   // Fliegendes Referenzieren aktivieren erkennen
   IF #FlyRef AND NOT #sbRefTypEdge THEN
     #sbRefTyp := True;
   END_IF;
   // Fliegendes Referenzieren aktivieren Flanke merken
   #sbRefTypEdge := #FlyRef;

   // Fliegendes Referenzieren Flankenmerker wieder zurücksetzen
   IF NOT #FlyRef THEN
     #sbRefTyp := False;
     #siRefTypCyc := 0;
   END_IF;

   // Betriebsart aktivieren erkennen (RQ 3901129, RQ 4094299)
   IF #ExecuteMode AND NOT #sbExecuteEdge THEN
     #sbExecute := True;
     #siExecuteCyc := 0;
   ELSIF #ActMode <> #ModePos THEN
     #sbExecute := FALSE;
   ELSIF #siExecuteCyc > (2 * #siCycWait) THEN
     IF #ModePos <> 4 THEN
       #sbExecute := FALSE;
     ELSE
       IF #sxRecvBuf.ZSW1.%X11 OR NOT #ExecuteMode THEN
         #sbExecute := FALSE;
       END_IF;
     END_IF;
   ELSE
     ; // not used
   END_IF;

   IF #siExecuteCyc > 100 THEN
     #siExecuteCyc := 0;
   ELSE
     #siExecuteCyc := #siExecuteCyc + 1;
   END_IF;

   // Verfahrauftrag aktivieren Flanke merken
   #sbExecuteEdge := #ExecuteMode;

   // Betriebsart MDI / Sollwertdirektvorgabe Flanke merken
   (*IF #sxSendBuf.sxEPosSTW1.MdiStart AND NOT #sbMdiStartEdge THEN
             #sbMdiStart := True;
         END_IF;
         // Betriebsart MDI / Sollwertdirektvorgabe Flanke merken
         #sbMdiStartEdge := #sxSendBuf.sxEPosSTW1.MdiStart AND NOT #Busy;*)

   // Verfahrauftragflankenmerker wieder zurücksetzen
   (*IF NOT #sxSendBuf.sxEPosSTW1.MdiStart THEN
             #sbMdiStart := False;
             #siMdiStartCyc := 0;
         END_IF;*)

   IF #sxSendBuf.EPosSTW1.%X15 AND NOT #sbMdiStartEdge THEN
     #sbMdiStart := True;
   END_IF;
   // Betriebsart MDI / Sollwertdirektvorgabe Flanke merken
   #sbMdiStartEdge := #sxSendBuf.EPosSTW1.%X15 AND NOT #sbBusy;

   // Verfahrauftragflankenmerker wieder zurücksetzen
   IF NOT #sxSendBuf.EPosSTW1.%X15 THEN
     #sbMdiStart := False;
     #siMdiStartCyc := 0;
   END_IF;

   // Schreibdaten zusammenstellen
   // Steuerword STW1 für alle Betriebsart aufbereiten
   (*#sxSendBuf.sxSTW1.RejTrvTsk        := #RejTrvTsk;
         #sxSendBuf.sxSTW1.IntMStop         := #IntMStop;
         #sxSendBuf.sxSTW1.AckFault         := #AckFlt;*)

   #sxSendBuf.STW1.%X4 := #CancelTraversing;
   #sxSendBuf.STW1.%X5 := #IntermediateStop;
   #sxSendBuf.STW1.%X7 := #AckError;
   #sxSendBuf.STW1.%X1 := TRUE;
   #sxSendBuf.STW1.%X2 := TRUE;
   #sxSendBuf.STW1.%X3 := TRUE;
   #sxSendBuf.STW1.%X10 := TRUE;

   // Hauptbetriebsart "Positionieren / manueller Sollwertvorgabe (MDI)" 
   // Betriebsart "Positionieren Relativ positiv" oder "Positionieren Relativ negativ"
   IF (#siModePos = 1 AND #sbModePos) THEN

     // Antrieb einschalten
     //#sxSendBuf.sxSTW1.Off1 := #sbOff1;
     #sxSendBuf.STW1.%X0 := #sbOff1;

     // nicht verwendete Signale für den 1. Schritt und eventuell weitere Schritte
     (*#sxSendBuf.sxSTW1.Jog1          := False;
             #sxSendBuf.sxSTW1.Jog2          := False;
             #sxSendBuf.sxEPosSTW1.MdiTyp    := False;
             #sxSendBuf.sxEPosSTW1.MdiPos    := False;
             #sxSendBuf.sxEPosSTW1.MdiNeg    := False;
             #sxSendBuf.sxEPosSTW1.MdiSetup  := False;
             #sxSendBuf.sxEPosSTW2.SetRefPt  := False;
             #sxSendBuf.sxEPosSTW2.JogInc    := False;
             #sxSendBuf.sxEPosSTW2.RefStDi   := False;
             #sxSendBuf.sxSTW1.RefStart      := False;
             #sxSendBuf.sxEPosSTW2.RefTyp    := False;
             #sxSendBuf.sxEPosSTW1.MdiStart  := False;*)
     #sxSendBuf.STW1.%X8 := False;
     #sxSendBuf.STW1.%X9 := False;
     #sxSendBuf.EPosSTW1.%X8 := False;
     #sxSendBuf.EPosSTW1.%X9 := False;
     #sxSendBuf.EPosSTW1.%X10 := False;
     #sxSendBuf.EPosSTW1.%X14 := False;
     #sxSendBuf.EPosSTW2.%X1 := False;
     #sxSendBuf.EPosSTW2.%X5 := False;
     #sxSendBuf.EPosSTW2.%X9 := False;
     #sxSendBuf.STW1.%X11 := False;
     #sxSendBuf.EPosSTW2.%X8 := False;
     #sxSendBuf.EPosSTW1.%X15 := False;


     // Nach dem Einschalten des Antriebes, prüfen ob der Antrieb betriebsbereit, in Operation ohne Fehler und Warnung ist, 
     // dann die Betriebsart MDI / Sollwertvorgabe Start gesetzt werden
     IF #sbOff1 AND #sbReady AND #sbIOp AND NOT #sbFault THEN

       // Betriebsart MDI / Sollwertdirektvorgabe setzen
       //#sxSendBuf.sxEPosSTW1.MdiStart := True;
       #sxSendBuf.EPosSTW1.%X15 := True;

       // Positioniertyp auf relatives Positionieren stellen 
       //#sxSendBuf.sxEPosSTW1.MdiTyp := False;
       #sxSendBuf.EPosSTW1.%X8 := False;

       // die Richtungswahl für das Positionieren auf positive Richtung oder negative Richtung einstellen
       IF #Positive AND NOT #Negative THEN

         // positive Richtung
         //#sxSendBuf.sxEPosSTW1.MdiPos := True;
         #sxSendBuf.EPosSTW1.%X9 := True;

         // negative Richtung
         //#sxSendBuf.sxEPosSTW1.MdiNeg := False;
         #sxSendBuf.EPosSTW1.%X10 := False;

         // die Richtungswahl für das Positionieren auf negative Richtung einstellen                
       ELSIF NOT #Positive AND #Negative THEN

         // positive Richtung
         //#sxSendBuf.sxEPosSTW1.MdiPos := False;
         #sxSendBuf.EPosSTW1.%X9 := False;

         // negative Richtung
         //#sxSendBuf.sxEPosSTW1.MdiNeg := True;
         #sxSendBuf.EPosSTW1.%X10 := True;

         // die Richtungswahl für das Positionieren auf keine Richtung einstellen                
       ELSE

         // positive Richtung
         //#sxSendBuf.sxEPosSTW1.MdiPos := False;
         #sxSendBuf.EPosSTW1.%X9 := False;

         // negative Richtung
         //#sxSendBuf.sxEPosSTW1.MdiNeg := False;
         #sxSendBuf.EPosSTW1.%X10 := False;

       END_IF;

       // Nach dem Einschalten des Antriebes und dem Betriebsart MDI / Sollwertvorgabe starten, 
       // ein Paar Zyklen warten bevor die Flanke für die Sollwertübernahme MDI gesetzt werden kann
       IF #sbMdiStart AND (#siMdiStartCyc < #siCycWait) THEN
         #siMdiStartCyc := #siMdiStartCyc + 1;
       ELSE
         // Flanke Sollwertübernahme MDI
         //#sxSendBuf.sxSTW1.TrvStart := #Execute;
         #sxSendBuf.STW1.%X6 := #sbExecute;

       END_IF;

       // "Fliegendes Referentieren" aktivieren
       // "Fliegendes Referenzieren" erst nach Einschalten des Antriebes möglich
       IF #sbRefTyp THEN

         // Referenziertyp auf "Fliegendes Referenzieren" einstellen
         //#sxSendBuf.sxEPosSTW2.RefTyp := True;
         #sxSendBuf.EPosSTW2.%X8 := True;

         // Nach der Anwahl des Referenziertyps "Fliegendes Referenzieren", 
         // ein Zyklus später kann das Referenzieren gestartet
         IF (#siRefTypCyc = 0) THEN
           #siRefTypCyc := #siRefTypCyc + 1;
         ELSE
           // Referenzieren starten
           //#sxSendBuf.sxSTW1.RefStart := True;
           #sxSendBuf.STW1.%X11 := True;

         END_IF;
       END_IF;
     END_IF;

     // Betriebsart "Positionieren Absolut" oder "Positonieren Absolut positiv" oder "Positionieren Absolut negativ"
   ELSIF #siModePos = 2 AND #sbModePos THEN

     // Antrieb einschalten
     //#sxSendBuf.sxSTW1.Off1 := #sbOff1;
     #sxSendBuf.STW1.%X0 := #sbOff1;

     // nicht verwendete Signale für den 1. Schritt und eventuell weitere Schritte
     (*#sxSendBuf.sxSTW1.Jog1         := False;
             #sxSendBuf.sxSTW1.Jog2         := False;
             #sxSendBuf.sxEPosSTW1.MdiTyp   := False;
             #sxSendBuf.sxEPosSTW1.MdiPos   := False;
             #sxSendBuf.sxEPosSTW1.MdiNeg   := False;
             #sxSendBuf.sxEPosSTW1.MdiSetup := False;
             #sxSendBuf.sxEPosSTW2.SetRefPt := False;
             #sxSendBuf.sxEPosSTW2.JogInc   := False;
             #sxSendBuf.sxEPosSTW2.RefStDi  := False;
             #sxSendBuf.sxSTW1.RefStart     := False;
             #sxSendBuf.sxEPosSTW2.RefTyp   := False;
             #sxSendBuf.sxEPosSTW1.MdiStart := False;*)
     #sxSendBuf.STW1.%X8 := False;
     #sxSendBuf.STW1.%X9 := False;
     #sxSendBuf.EPosSTW1.%X8 := False;
     #sxSendBuf.EPosSTW1.%X9 := False;
     #sxSendBuf.EPosSTW1.%X10 := False;
     #sxSendBuf.EPosSTW1.%X14 := False;
     #sxSendBuf.EPosSTW2.%X1 := False;
     #sxSendBuf.EPosSTW2.%X5 := False;
     #sxSendBuf.EPosSTW2.%X9 := False;
     #sxSendBuf.STW1.%X11 := False;
     #sxSendBuf.EPosSTW2.%X8 := False;
     #sxSendBuf.EPosSTW1.%X15 := False;

     // Nach dem Einschalten des Antriebes, prüfen ob der Antrieb betriebsbereit, in Operation ohne Fehler und Warnung ist, 
     // dann die Betriebsart MDI / Sollwertvorgabe Start gesetzt werden
     IF #sbOff1 AND #sbReady AND #sbIOp AND NOT #sbFault THEN

       // Betriebsart MDI / Sollwertdirektvorgabe setzen
       //#sxSendBuf.sxEPosSTW1.MdiStart := True;
       #sxSendBuf.EPosSTW1.%X15 := True;

       // Positioniertyp auf absolutes Positionieren stellen 
       //#sxSendBuf.sxEPosSTW1.MdiTyp := True;
       #sxSendBuf.EPosSTW1.%X8 := True;

       // die Richtungswahl für das Positionieren auf positive Richtung oder negative Richtung einstellen
       IF #Positive AND NOT #Negative THEN

         // positive Richtung
         //#sxSendBuf.sxEPosSTW1.MdiPos := True;
         #sxSendBuf.EPosSTW1.%X9 := True;

         // negative Richtung
         //#sxSendBuf.sxEPosSTW1.MdiNeg := False;
         #sxSendBuf.EPosSTW1.%X10 := False;

         // die Richtungswahl für das Positionieren auf negative Richtung einstellen                
       ELSIF NOT #Positive AND #Negative THEN

         // positive Richtung
         //#sxSendBuf.sxEPosSTW1.MdiPos := False;
         #sxSendBuf.EPosSTW1.%X9 := False;

         // negative Richtung
         //#sxSendBuf.sxEPosSTW1.MdiNeg := True;
         #sxSendBuf.EPosSTW1.%X10 := True;

         // die Richtungswahl für das Positionieren auf keine Richtung einstellen                
       ELSE

         // positive Richtung
         //#sxSendBuf.sxEPosSTW1.MdiPos := False;
         #sxSendBuf.EPosSTW1.%X9 := False;

         // negative Richtung
         //#sxSendBuf.sxEPosSTW1.MdiNeg := False;
         #sxSendBuf.EPosSTW1.%X10 := False;

       END_IF;

       // Nach dem Einschalten des Antriebes und dem Betriebsart MDI / Sollwertvorgabe starten, 
       // ein Paar Zyklen warten bevor die Flanke für die Sollwertübernahme MDI gesetzt werden kann
       IF #sbMdiStart AND (#siMdiStartCyc < #siCycWait) THEN
         #siMdiStartCyc := #siMdiStartCyc + 1;
       ELSE
         // Flanke Sollwertübernahme MDI
         //#sxSendBuf.sxSTW1.TrvStart := #Execute;
         #sxSendBuf.STW1.%X6 := #sbExecute;

       END_IF;

       // "Fliegendes Referentieren" aktivieren
       // "Fliegendes Referenzieren" erst nach Einschalten des Antriebes möglich
       IF #sbRefTyp THEN

         // Referenziertyp auf "Fliegendes Referenzieren" einstellen
         //#sxSendBuf.sxEPosSTW2.RefTyp := True;
         #sxSendBuf.EPosSTW2.%X8 := True;

         // Nach der Anwahl des Referenziertyps "Fliegendes Referenzieren", 
         // ein Zyklus später kann das Referenzieren gestartet
         IF (#siRefTypCyc = 0) THEN
           #siRefTypCyc := #siRefTypCyc + 1;
         ELSE
           // Referenzieren starten
           //#sxSendBuf.sxSTW1.RefStart := True;
           #sxSendBuf.STW1.%X11 := True;

         END_IF;
       END_IF;
     END_IF;

     // Betriebsart "Positionieren als Einrichten positiv" oder "Positionieren als Einrichten negativ"
   ELSIF #siModePos = 3 AND #sbModePos THEN

     // Antrieb einschalten
     //#sxSendBuf.sxSTW1.Off1 := #sbOff1;
     #sxSendBuf.STW1.%X0 := #sbOff1;

     // nicht verwendete Signale für den 1. Schritt und eventuell weitere Schritte
     (*#sxSendBuf.sxSTW1.Jog1           := False;
             #sxSendBuf.sxSTW1.Jog2           := False;
             #sxSendBuf.sxEPosSTW1.MdiTyp     := False;
             #sxSendBuf.sxEPosSTW1.MdiPos     := False;
             #sxSendBuf.sxEPosSTW1.MdiNeg     := False;
             #sxSendBuf.sxEPosSTW1.MdiSetup   := False;
             #sxSendBuf.sxEPosSTW2.SetRefPt   := False;
             #sxSendBuf.sxEPosSTW2.JogInc     := False;
             #sxSendBuf.sxEPosSTW2.RefStDi    := False;
             #sxSendBuf.sxSTW1.RefStart       := False;
             #sxSendBuf.sxEPosSTW2.RefTyp     := False;
             #sxSendBuf.sxEPosSTW1.MdiStart   := False;*)
     #sxSendBuf.STW1.%X8 := False;
     #sxSendBuf.STW1.%X9 := False;
     #sxSendBuf.EPosSTW1.%X8 := False;
     #sxSendBuf.EPosSTW1.%X9 := False;
     #sxSendBuf.EPosSTW1.%X10 := False;
     #sxSendBuf.EPosSTW1.%X14 := False;
     #sxSendBuf.EPosSTW2.%X1 := False;
     #sxSendBuf.EPosSTW2.%X5 := False;
     #sxSendBuf.EPosSTW2.%X9 := False;
     #sxSendBuf.STW1.%X11 := False;
     #sxSendBuf.EPosSTW2.%X8 := False;
     #sxSendBuf.EPosSTW1.%X15 := False;

     // Nach dem Einschalten des Antriebes, prüfen ob der Antrieb betriebsbereit, in Operation ohne Fehler und Warnung ist, 
     // dann die Betriebsart MDI / Sollwertvorgabe Start gesetzt werden
     IF #sbOff1 AND #sbReady AND #sbIOp AND NOT #sbFault THEN

       // Betriebsart MDI / Sollwertdirektvorgabe setzen
       //#sxSendBuf.sxEPosSTW1.MdiStart := True;
       #sxSendBuf.EPosSTW1.%X15 := True;

       // Positioniertyp auf absolutes Positionieren stellen 
       //#sxSendBuf.sxEPosSTW1.MdiTyp := True;
       #sxSendBuf.EPosSTW1.%X8 := True;

       // die Anwahl für MDI Modus auf Einrichten einstellen
       //#sxSendBuf.sxEPosSTW1.MdiSetup := True;
       #sxSendBuf.EPosSTW1.%X14 := True;

       // die Richtungswahl für das Positionieren auf positive Richtung oder negative Richtung einstellen
       IF #Positive AND NOT #Negative THEN

         // positive Richtung
         //#sxSendBuf.sxEPosSTW1.MdiPos := True;
         #sxSendBuf.EPosSTW1.%X9 := True;

         // negative Richtung
         //#sxSendBuf.sxEPosSTW1.MdiNeg := False;
         #sxSendBuf.EPosSTW1.%X10 := False;

         // die Richtungswahl für das Positionieren auf negative Richtung einstellen                
       ELSIF NOT #Positive AND #Negative THEN

         // positive Richtung
         //#sxSendBuf.sxEPosSTW1.MdiPos := False;
         #sxSendBuf.EPosSTW1.%X9 := False;

         // negative Richtung
         //#sxSendBuf.sxEPosSTW1.MdiNeg := True;
         #sxSendBuf.EPosSTW1.%X10 := True;

         // die Richtungswahl für das Positionieren auf keine Richtung einstellen                
       ELSE

         // positive Richtung
         //#sxSendBuf.sxEPosSTW1.MdiPos := False;
         #sxSendBuf.EPosSTW1.%X9 := False;

         // negative Richtung
         //#sxSendBuf.sxEPosSTW1.MdiNeg := False;
         #sxSendBuf.EPosSTW1.%X10 := False;

       END_IF;

       // Nach dem Einschalten des Antriebes und dem Betriebsart MDI / Sollwertvorgabe starten, 
       // ein Paar Zyklen warten bevor die Flanke für die Sollwertübernahme MDI gesetzt werden kann
       IF #sbMdiStart AND (#siMdiStartCyc < #siCycWait) THEN
         #siMdiStartCyc := #siMdiStartCyc + 1;
       ELSE
         // Flanke Sollwertübernahme MDI
         //#sxSendBuf.sxSTW1.TrvStart := #Execute;
         #sxSendBuf.STW1.%X6 := #sbExecute;

       END_IF;

       // "Fliegendes Referentieren" aktivieren
       // "Fliegendes Referenzieren" erst nach Einschalten des Antriebes möglich
       IF #sbRefTyp THEN

         // Referenziertyp auf "Fliegendes Referenzieren" einstellen
         //#sxSendBuf.sxEPosSTW2.RefTyp := True;
         #sxSendBuf.EPosSTW2.%X8 := True;

         // Nach der Anwahl des Referenziertyps "Fliegendes Referenzieren", 
         // ein Zyklus später kann das Referenzieren gestartet
         IF (#siRefTypCyc = 0) THEN
           #siRefTypCyc := #siRefTypCyc + 1;
         ELSE
           // Referenzieren starten
           //#sxSendBuf.sxSTW1.RefStart := True;
           #sxSendBuf.STW1.%X11 := True;

         END_IF;
       END_IF;
     END_IF;

     // Hauptbetriebsart "Referenzieren" (Reference)
     // Betriebsart "Referenzieren - Referenzpunktfahrt positiv" oder "Referenzieren - Referenzpunktfahrt negativ"
   ELSIF #siModePos = 4 AND #sbModePos THEN

     // Antrieb einschalten
     //#sxSendBuf.sxSTW1.Off1 := #sbOff1;
     #sxSendBuf.STW1.%X0 := #sbOff1;

     // nicht verwendete Signale für den 1. Schritt und eventuell weitere Schritte
     (*#sxSendBuf.sxSTW1.Jog1         := False;
             #sxSendBuf.sxSTW1.Jog2         := False;
             #sxSendBuf.sxEPosSTW1.MdiStart := False;
             #sxSendBuf.sxEPosSTW2.SetRefPt := False;
             #sxSendBuf.sxEPosSTW2.JogInc   := False;
             #sxSendBuf.sxEPosSTW2.RefTyp   := False;
             #sxSendBuf.sxSTW1.RefStart     := False;
             #sxSendBuf.sxEPosSTW2.RefStDi  := False;*)
     #sxSendBuf.STW1.%X8 := False;
     #sxSendBuf.STW1.%X9 := False;
     #sxSendBuf.EPosSTW1.%X15 := False;
     #sxSendBuf.EPosSTW2.%X1 := False;
     #sxSendBuf.EPosSTW2.%X5 := False;
     #sxSendBuf.EPosSTW2.%X8 := False;
     #sxSendBuf.STW1.%X11 := False;
     #sxSendBuf.EPosSTW2.%X9 := False;

     // Nach dem Einschalten des Antriebes, prüfen ob der Antrieb betriebsbereit, in Operation ohne Fehler und Warnung ist, 
     // dann die Betriebsart MDI / Sollwertvorgabe Start gesetzt werden
     IF #sbOff1 AND #sbReady AND #sbIOp AND NOT #sbFault THEN

       // Referenzieren starten
       //#sxSendBuf.sxSTW1.RefStart := #Execute;
       #sxSendBuf.STW1.%X11 := #sbExecute;

       // die Richtungswahl für das Referenzpunktfahrt positiv einstellen
       IF #Positive AND NOT #Negative THEN

         // positive Referenzpunktfahrt
         //#sxSendBuf.sxEPosSTW2.RefStDi := False;
         #sxSendBuf.EPosSTW2.%X9 := False;

         // die Richtungswahl für das Referenzpunktfahrt negativ einstellen                
       ELSIF NOT #Positive AND #Negative THEN

         // negative Referenzpunktfahrt
         //#sxSendBuf.sxEPosSTW2.RefStDi := True;
         #sxSendBuf.EPosSTW2.%X9 := True;

       END_IF;
     END_IF;

     // Betriebsart "Referenzieren - Referenzpunkt setzen"
   ELSIF #siModePos = 5 AND #sbModePos THEN

     // Antrieb einschalten
     //#sxSendBuf.sxSTW1.Off1 := #sbOff1;
     #sxSendBuf.STW1.%X0 := #sbOff1;

     // nicht verwendete Signale für den 1. Schritt und eventuell weitere Schritte
     (*#sxSendBuf.sxSTW1.Jog1          := False;
             #sxSendBuf.sxSTW1.Jog2          := False;
             #sxSendBuf.sxSTW1.RefStart      := False;
             #sxSendBuf.sxEPosSTW1.MdiStart  := False;
             #sxSendBuf.sxEPosSTW2.JogInc    := False;
             #sxSendBuf.sxEPosSTW2.RefTyp    := False;
             #sxSendBuf.sxEPosSTW2.RefStDi   := False;
             #sxSendBuf.sxEPosSTW2.SetRefPt  := False;*)
     #sxSendBuf.STW1.%X8 := False;
     #sxSendBuf.STW1.%X9 := False;
     #sxSendBuf.STW1.%X11 := False;
     #sxSendBuf.EPosSTW1.%X15 := False;
     #sxSendBuf.EPosSTW2.%X5 := False;
     #sxSendBuf.EPosSTW2.%X8 := False;
     #sxSendBuf.EPosSTW2.%X9 := False;
     #sxSendBuf.EPosSTW2.%X1 := False;

     // Nach dem Einschalten des Antriebes, prüfen ob der Antrieb betriebsbereit, in Operation ohne Fehler und Warnung ist, 
     // dann die Betriebsart MDI / Sollwertvorgabe Start gesetzt werden
     IF NOT #sbFault THEN

       // Referenzpunktfahrt negativ
       //#sxSendBuf.sxEPosSTW2.SetRefPt := #Execute;
       #sxSendBuf.EPosSTW2.%X1 := #sbExecute;

     END_IF;

     // Hauptbetriebsart "Verfahrsätze" (Traversing Blocks)
   ELSIF #siModePos = 6 AND #sbModePos THEN

     // Antrieb einschalten
     //#sxSendBuf.sxSTW1.Off1 := #sbOff1;
     #sxSendBuf.STW1.%X0 := #sbOff1;

     // nicht verwendete Signale für den 1. Schritt und eventuell weitere Schritte
     (*#sxSendBuf.sxSTW1.Jog1          := False;
             #sxSendBuf.sxSTW1.Jog2          := False;
             #sxSendBuf.sxEPosSTW1.MdiTyp    := False;
             #sxSendBuf.sxEPosSTW1.MdiPos    := False;
             #sxSendBuf.sxEPosSTW1.MdiNeg    := False;
             #sxSendBuf.sxEPosSTW1.MdiSetup  := False;
             #sxSendBuf.sxEPosSTW2.SetRefPt  := False;
             #sxSendBuf.sxEPosSTW2.JogInc    := False;
             #sxSendBuf.sxEPosSTW2.RefStDi   := False;
             #sxSendBuf.sxEPosSTW2.RefTyp    := False;
             #sxSendBuf.sxSTW1.RefStart      := False;
             #sxSendBuf.sxEPosSTW1.TrvBit0   := False;
             #sxSendBuf.sxEPosSTW1.TrvBit1   := False;
             #sxSendBuf.sxEPosSTW1.TrvBit2   := False;
             #sxSendBuf.sxEPosSTW1.TrvBit3   := False;
             #sxSendBuf.sxEPosSTW1.TrvBit4   := False;
             #sxSendBuf.sxEPosSTW1.TrvBit5   := False;
             #sxSendBuf.sxEPosSTW1.MdiStart  := False;*)
     #sxSendBuf.STW1.%X8 := False;
     #sxSendBuf.STW1.%X9 := False;
     #sxSendBuf.EPosSTW1.%X8 := False;
     #sxSendBuf.EPosSTW1.%X9 := False;
     #sxSendBuf.EPosSTW1.%X10 := False;
     #sxSendBuf.EPosSTW1.%X14 := False;
     #sxSendBuf.EPosSTW2.%X1 := False;
     #sxSendBuf.EPosSTW2.%X5 := False;
     #sxSendBuf.EPosSTW2.%X9 := False;
     #sxSendBuf.EPosSTW2.%X8 := False;
     #sxSendBuf.STW1.%X11 := False;
     #sxSendBuf.EPosSTW1.%X0 := False;
     #sxSendBuf.EPosSTW1.%X1 := False;
     #sxSendBuf.EPosSTW1.%X2 := False;
     #sxSendBuf.EPosSTW1.%X3 := False;
     #sxSendBuf.EPosSTW1.%X4 := False;
     #sxSendBuf.EPosSTW1.%X5 := False;
     #sxSendBuf.EPosSTW1.%X15 := False;

     // Bei der Auswahl der Verfahrsätze entspricht die Position der Verfahrensatznummer 
     // Verfahrsatznummer aus der Position ermitteln und in die einzelnen Bit's aufteilen
     // Es sind die Verfahrsatznummern 0 - 63 möglich
     IF (DINT_TO_INT(#Position) < 0) OR (DINT_TO_INT(#Position) > 63) THEN
       // Fehler, ungültiger Verfahrsatznummer
       #swStatus := 16#8204;
       #Error := True;
     ELSE
       // Fehler wieder zurücknehmen, wenn er mal ausgelöst wurde
       IF #swStatus = 16#8204 THEN
         #swStatus := 16#7002;
         #Error := False;
       END_IF;

       // Verfahrsatznummer Bit 0 ermitteln
       IF (DINT_TO_WORD(#Position) AND W#16#01) = W#16#01 THEN
         //#sxSendBuf.sxEPosSTW1.TrvBit0 := True;
         #sxSendBuf.EPosSTW1.%X0 := True;
       END_IF;

       // Verfahrsatznummer Bit 1 ermitteln
       IF (DINT_TO_WORD(#Position) AND W#16#02) = W#16#02 THEN
         //#sxSendBuf.sxEPosSTW1.TrvBit1 := True;
         #sxSendBuf.EPosSTW1.%X1 := True;
       END_IF;

       // Verfahrsatznummer Bit 2 ermitteln
       IF (DINT_TO_WORD(#Position) AND W#16#04) = W#16#04 THEN
         //#sxSendBuf.sxEPosSTW1.TrvBit2 := True;
         #sxSendBuf.EPosSTW1.%X2 := True;
       END_IF;

       // Verfahrsatznummer Bit 3 ermitteln
       IF (DINT_TO_WORD(#Position) AND W#16#08) = W#16#08 THEN
         //#sxSendBuf.sxEPosSTW1.TrvBit3 := True;
         #sxSendBuf.EPosSTW1.%X3 := True;
       END_IF;

       // Verfahrsatznummer Bit 4 ermitteln
       IF (DINT_TO_WORD(#Position) AND W#16#10) = W#16#10 THEN
         //#sxSendBuf.sxEPosSTW1.TrvBit4 := True;
         #sxSendBuf.EPosSTW1.%X4 := True;
       END_IF;

       // Verfahrsatznummer Bit 5 ermitteln
       IF (DINT_TO_WORD(#Position) AND W#16#20) = W#16#20 THEN
         //#sxSendBuf.sxEPosSTW1.TrvBit5 := True;
         #sxSendBuf.EPosSTW1.%X5 := True;
       END_IF;

       // Nach dem Einschalten des Antriebes, prüfen ob der Antrieb betriebsbereit, in Operation ohne Fehler und Warnung ist, 
       // dann die Betriebsart MDI / Sollwertvorgabe Start gesetzt werden
       IF #sbOff1 AND #sbReady AND #sbIOp AND NOT #sbFault THEN

         #sxSendBuf.STW1.%X6 := #sbExecute;

         // "Fliegendes Referentieren" aktivieren
         // "Fliegendes Referenzieren" erst nach Einschalten des Antriebes möglich
         IF #sbRefTyp THEN

           // Referenziertyp auf "Fliegendes Referenzieren" einstellen
           //#sxSendBuf.sxEPosSTW2.RefTyp := True;
           #sxSendBuf.EPosSTW2.%X8 := True;

           // Nach der Anwahl des Referenziertyps "Fliegendes Referenzieren", 
           // ein Zyklus später kann das Referenzieren gestartet
           IF (#siRefTypCyc = 0) THEN
             #siRefTypCyc := #siRefTypCyc + 1;
           ELSE
             // Referenzieren starten
             //#sxSendBuf.sxSTW1.RefStart := True;
             #sxSendBuf.STW1.%X11 := True;
           END_IF;
         END_IF;
       END_IF;
     END_IF;

     // Hauptbetriebsart "Tippen" (Jogging)
     // Betriebsart "Tippen positiv" oder "Tippen negativ" angewählt 
   ELSIF #siModePos = 7 AND #sbModePos THEN

     // Antrieb einschalten
     //#sxSendBuf.sxSTW1.Off1 := #sbOff1;
     #sxSendBuf.STW1.%X0 := #sbOff1;

     // nicht verwendete Signale für den 1. Schritt und eventuell weitere Schritte
     (*#sxSendBuf.sxEPosSTW1.MdiStart := False;
             #sxSendBuf.sxEPosSTW2.JogInc   := False;
             #sxSendBuf.sxSTW1.Jog1         := False;
             #sxSendBuf.sxSTW1.Jog2         := False;
             #sxSendBuf.sxEPosSTW2.RefTyp   := False;
             #sxSendBuf.sxSTW1.RefStart     := False;
             #sxSendBuf.sxEPosSTW2.SetRefPt  := False;*)

     #sxSendBuf.EPosSTW1.%X15 := False;
     #sxSendBuf.EPosSTW2.%X5 := False;
     #sxSendBuf.STW1.%X8 := False;
     #sxSendBuf.STW1.%X9 := False;
     #sxSendBuf.EPosSTW2.%X8 := False;
     #sxSendBuf.STW1.%X11 := False;
     #sxSendBuf.EPosSTW2.%X1 := False;

     // Nach dem Einschalten des Antriebes, prüfen ob der Antrieb betriebsbereit, in Operation ohne Fehler und Warnung ist, 
     // dann kann Tippen positiv oder negativ gesetzt werden
     IF #sbOff1 AND #sbReady AND #sbIOp AND NOT #sbFault THEN

       // Tippen positiv
       IF #Jog1 AND NOT #Jog2 THEN
         //#sxSendBuf.sxSTW1.Jog1 := True;
         #sxSendBuf.STW1.%X8 := True;
       END_IF;

       // Tippen negativ
       IF #Jog2 AND NOT #Jog1 THEN
         //#sxSendBuf.sxSTW1.Jog2 := True;
         #sxSendBuf.STW1.%X9 := True;
       END_IF;

       // "Fliegendes Referentieren" aktivieren
       // "Fliegendes Referenzieren" erst nach Einschalten des Antriebes möglich
       IF #sbRefTyp THEN

         // Referenziertyp auf "Fliegendes Referenzieren" einstellen
         //#sxSendBuf.sxEPosSTW2.RefTyp := #FlyRef;
         #sxSendBuf.EPosSTW2.%X8 := #FlyRef;

         // Nach der Anwahl des Referenziertyps "Fliegendes Referenzieren", 
         // ein Zyklus später kann das Referenzieren gestartet
         IF (#siRefTypCyc = 0) THEN
           #siRefTypCyc := #siRefTypCyc + 1;
         ELSE
           // Referenzieren starten
           //#sxSendBuf.sxSTW1.RefStart := True;
           #sxSendBuf.STW1.%X11 := True;
         END_IF;
       END_IF;
     END_IF;

     // Betriebsart "Tippen positiv / Tippen negativ inkrementell" 
   ELSIF #siModePos = 8 AND #sbModePos THEN

     // Antrieb einschalten
     //#sxSendBuf.sxSTW1.OFF1 := #sbOff1;
     #sxSendBuf.STW1.%X0 := #sbOff1;

     // nicht verwendete Signale für den 1. Schritt und eventuell weitere Schritte
     (*#sxSendBuf.sxEPosSTW1.MdiStart := False;
             #sxSendBuf.sxEPosSTW2.JogInc   := False;
             #sxSendBuf.sxSTW1.Jog1         := False;
             #sxSendBuf.sxSTW1.Jog2         := False;
             #sxSendBuf.sxSTW1.RefStart     := False;
             #sxSendBuf.sxEPosSTW2.RefTyp   := False;
             #sxSendBuf.sxEPosSTW2.SetRefPt  := False;*)

     #sxSendBuf.EPosSTW1.%X15 := False;
     #sxSendBuf.EPosSTW2.%X5 := False;
     #sxSendBuf.STW1.%X8 := False;
     #sxSendBuf.STW1.%X9 := False;
     #sxSendBuf.STW1.%X11 := False;
     #sxSendBuf.EPosSTW2.%X8 := False;
     #sxSendBuf.EPosSTW2.%X1 := False;

     // Nach dem Einschalten des Antriebes, ein Paar Zyklen warten bevor Tippen negativ gesetzt werden kann
     // Nach dem Einschalten des Antriebes, prüfen ob der Antrieb betriebsbereit, in Operation ohne Fehler und Warnung ist, 
     // dann kann Tippen positiv oder negativ gesetzt werden
     IF #sbOff1 AND #sbReady AND #sbIOp AND NOT #sbFault THEN

       // Tippen inkrementell einstellen
       //#sxSendBuf.sxEPosSTW2.JogInc := True;
       #sxSendBuf.EPosSTW2.%X5 := True;

       #sbJogInc := True;

       // Nach dem Einstellen des Antriebes, ein Paar Zyklen warten bevor Tippen negativ oder Tippen positiv gesetz werden kann
       IF #sbJogInc AND (#siJogIncCyc = 0) THEN
         #siJogIncCyc := #siJogIncCyc + 1;
       ELSE

         // Tippen positiv oder negativ inkrementell zulassen
         IF #Jog1 XOR #Jog2 THEN

           //#sxSendBuf.sxSTW1.Jog1 := #Jog1;
           //#sxSendBuf.sxSTW1.Jog2 := #Jog2;
           #sxSendBuf.STW1.%X8 := #Jog1;
           #sxSendBuf.STW1.%X9 := #Jog2;
         END_IF;
       END_IF;

       // "Fliegendes Referentieren" aktivieren
       // "Fliegendes Referenzieren" erst nach Einschalten des Antriebes möglich
       IF #sbRefTyp THEN

         // Referenziertyp auf "Fliegendes Referenzieren" einstellen
         //#sxSendBuf.sxEPosSTW2.RefTyp := True;
         #sxSendBuf.EPosSTW2.%X8 := True;

         // Nach der Anwahl des Referenziertyps "Fliegendes Referenzieren", 
         // ein Zyklus später kann das Referenzieren gestartet
         IF (#siRefTypCyc = 0) THEN
           #siRefTypCyc := #siRefTypCyc + 1;
         ELSE
           // Referenzieren starten
           //#sxSendBuf.sxSTW1.RefStart := True;
           #sxSendBuf.STW1.%X11 := True;
         END_IF;
       END_IF;
     END_IF;
   ELSE
     // Werte wieder zurücknehmen
     (*#sxSendBuf.sxSTW1.Off1          := #Off1;
             #sxSendBuf.sxSTW1.RejTrvTsk     := False;
             #sxSendBuf.sxSTW1.TrvStart      := False;
             #sxSendBuf.sxEPosSTW1.MdiStart  := False;
             #sxSendBuf.sxSTW1.Jog1          := False;
             #sxSendBuf.sxSTW1.Jog2          := False;
             #sxSendBuf.sxEPosSTW1.MdiTyp    := False;
             #sxSendBuf.sxEPosSTW1.MdiPos    := False;
             #sxSendBuf.sxEPosSTW1.MdiNeg    := False;
             #sxSendBuf.sxEPosSTW1.MdiTrTyp  := False;
             #sxSendBuf.sxEPosSTW1.MdiSetup  := False;
             #sxSendBuf.sxEPosSTW2.SetRefPt  := False;
             #sxSendBuf.sxEPosSTW2.RefTyp    := False;
             #sxSendBuf.sxEPosSTW2.RefStDi   := False;
             #sxSendBuf.sxEPosSTW2.JogInc    := False;
             #sxSendBuf.sxSTW1.RefStart      := False;*)

     #sxSendBuf.STW1.%X0 := #EnableAxis;
     #sxSendBuf.STW1.%X4 := False;
     #sxSendBuf.STW1.%X6 := False;
     #sxSendBuf.EPosSTW1.%X15 := False;
     #sxSendBuf.STW1.%X8 := False;
     #sxSendBuf.STW1.%X9 := False;
     #sxSendBuf.EPosSTW1.%X8 := False;
     #sxSendBuf.EPosSTW1.%X9 := False;
     #sxSendBuf.EPosSTW1.%X10 := False;
     #sxSendBuf.EPosSTW1.%X12 := False;
     #sxSendBuf.EPosSTW1.%X14 := False;
     #sxSendBuf.EPosSTW2.%X1 := False;
     #sxSendBuf.EPosSTW2.%X8 := False;
     #sxSendBuf.EPosSTW2.%X9 := False;
     #sxSendBuf.EPosSTW2.%X5 := False;
     #sxSendBuf.STW1.%X11 := False;
   END_IF; // Hauptbetriebsart "Verfahrsätze" (Traversing Blocks)

   //Den Eingang ConfigEPos auf die einzelnen Bits im Telegramm verschalten
   #sxSendBuf.STW1.%X1 := #ConfigEPos.%X0;
   #sxSendBuf.STW1.%X2 := #ConfigEPos.%X1;
   #sxSendBuf.EPosSTW2.%X14 := #ConfigEPos.%X2;
   #sxSendBuf.EPosSTW2.%X15 := #ConfigEPos.%X3;
   #sxSendBuf.EPosSTW2.%X11 := #ConfigEPos.%X4;
   #sxSendBuf.EPosSTW2.%X10 := #ConfigEPos.%X5;
   #sxSendBuf.EPosSTW2.%X2 := #ConfigEPos.%X6;
   #sxSendBuf.STW1.%X13 := #ConfigEPos.%X7;
   #sxSendBuf.EPosSTW1.%X12 := #ConfigEPos.%X8;
   #sxSendBuf.STW2.%X0 := #ConfigEPos.%X9;
   #sxSendBuf.STW2.%X1 := #ConfigEPos.%X10;
   #sxSendBuf.STW2.%X2 := #ConfigEPos.%X11;
   #sxSendBuf.STW2.%X3 := #ConfigEPos.%X12;
   #sxSendBuf.STW2.%X4 := #ConfigEPos.%X13;
   #sxSendBuf.STW2.%X7 := #ConfigEPos.%X14;
   #sxSendBuf.STW1.%X12 := #ConfigEPos.%X15;
   #sxSendBuf.STW1.%X14 := #ConfigEPos.%X16;
   #sxSendBuf.STW1.%X15 := #ConfigEPos.%X17;
   #sxSendBuf.EPosSTW1.%X6 := #ConfigEPos.%X18;
   #sxSendBuf.EPosSTW1.%X7 := #ConfigEPos.%X19;
   #sxSendBuf.EPosSTW1.%X11 := #ConfigEPos.%X20;
   #sxSendBuf.EPosSTW1.%X13 := #ConfigEPos.%X21;
   #sxSendBuf.EPosSTW2.%X3 := #ConfigEPos.%X22;
   #sxSendBuf.EPosSTW2.%X4 := #ConfigEPos.%X23;
   #sxSendBuf.EPosSTW2.%X6 := #ConfigEPos.%X24;
   #sxSendBuf.EPosSTW2.%X7 := #ConfigEPos.%X25;
   #sxSendBuf.EPosSTW2.%X12 := #ConfigEPos.%X26;
   #sxSendBuf.EPosSTW2.%X13 := #ConfigEPos.%X27;
   #sxSendBuf.STW2.%X5 := #ConfigEPos.%X28;
   #sxSendBuf.STW2.%X6 := #ConfigEPos.%X29;
   #sxSendBuf.STW2.%X8 := #ConfigEPos.%X30;
   #sxSendBuf.STW2.%X9 := #ConfigEPos.%X31;


   #swSendBuf[0] := #sxSendBuf.STW1;
   #swSendBuf[1] := #sxSendBuf.EPosSTW1;
   #swSendBuf[2] := #sxSendBuf.EPosSTW2;
   #swSendBuf[3] := #sxSendBuf.STW2;
   #swSendBuf[4] := #sxSendBuf.OverrideV;
   #swSendBuf[5] := #sxSendBuf.Position.%W1;
   #swSendBuf[6] := #sxSendBuf.Position.%W0;
   #swSendBuf[7] := #sxSendBuf.Velocity.%W1;
   #swSendBuf[8] := #sxSendBuf.Velocity.%W0;
   #swSendBuf[9] := #sxSendBuf.OverrideA;
   #swSendBuf[10] := #sxSendBuf.OverrideD;
   #swSendBuf[11] := #sxSendBuf.Reserve;

   //Prozessdaten zur Signalbaugruppe schreiben
   #piRetSFC := DPWR_DAT(LADDR := #HWIDSTW,
                         RECORD := #swSendBuf);

   // Fehler der Rückmeldung ausgeben
   #DiagID := INT_TO_WORD(#piRetSFC);

   //kein Fehler beim Schreiben
   IF #piRetSFC = 0 THEN

     // Fehler wieder zurück nehmen
     IF (#swStatus = 16#8601) THEN
       #swStatus := 16#7002;
       #Error := False;
     END_IF;

     //Prozessdaten von der Signalbaugruppe lesen
     #piRetSFC := DPRD_DAT(LADDR := #HWIDZSW,
                           RECORD => #swRecvBuf);

     // Fehlermeldung der Rückmeldung ausgeben
     #DiagID := INT_TO_WORD(#piRetSFC);

     //Fehler beim Lesen (Profibus-Kommunikation unterbrochen)
     IF #piRetSFC <> 0 THEN

       // Fehler
       #Error := TRUE;
       #swStatus := 16#8600;

       // Zustandsworte löschen
       #sxRecvBuf.ZSW1 := W#16#0;
       #sxRecvBuf.EPosZSW1 := W#16#0;
       #sxRecvBuf.EPosZSW2 := W#16#0;
       #sxRecvBuf.ZSW2 := W#16#0;
       #sxRecvBuf.NotUsed := W#16#00;
       #sxRecvBuf.Position := DW#16#00;
       #sxRecvBuf.Velocity := DW#16#00;
       #sxRecvBuf.ErrNr := W#16#00;
       #sxRecvBuf.WarnNr := W#16#00;
       #sxRecvBuf.Reserve := W#16#00;

       // Werte auslesen
     ELSE

       // Fehler wieder zurück nehmen
       IF (#swStatus = 16#8600) THEN
         #swStatus := 16#7002;
         #Error := False;
       END_IF;

       #sxRecvBuf.ZSW1 := #swRecvBuf[0];
       #sxRecvBuf.EPosZSW1 := #swRecvBuf[1];
       #sxRecvBuf.EPosZSW2 := #swRecvBuf[2];
       #sxRecvBuf.ZSW2 := #swRecvBuf[3];
       #sxRecvBuf.NotUsed := #swRecvBuf[4];
       #sxRecvBuf.Position.%W1 := #swRecvBuf[5];
       #sxRecvBuf.Position.%W0 := #swRecvBuf[6];
       #sxRecvBuf.Velocity.%W1 := #swRecvBuf[7];
       #sxRecvBuf.Velocity.%W0 := #swRecvBuf[8];
       #sxRecvBuf.ErrNr := #swRecvBuf[9];
       #sxRecvBuf.WarnNr := #swRecvBuf[10];
       #sxRecvBuf.Reserve := #swRecvBuf[11];

       // ZSW1 aufbereiten
       //#Busy := #sxRecvBuf.sxZSW1.IOp;
       #sbBusy := #sxRecvBuf.ZSW1.%X2;

       // Fehler auswerten
       IF #sxRecvBuf.ZSW1.%X3 THEN
         #swStatus := 16#8401;
         #Error := True;
       ELSIF #sxRecvBuf.ZSW1.%X6 THEN
         #swStatus := 16#8402;
         #Error := True;
       ELSE
         // Fehler wieder zurück nehmen
         IF (#swStatus = 16#8401) OR (#swStatus = 16#8402) THEN
           #swStatus := 16#7002;
           #Error := False;
         END_IF;
       END_IF;

       // EPOS_ZSW1            
       // EPOS-Wort-1 BIT 00 --> 1 = Active traversing block bit 0
       //IF #sxRecvBuf.sxEPosZSW1.ActTrvBit0 THEN
       IF #sxRecvBuf.EPosZSW1.%X0 THEN
         #swEPosZSW1 := #swEPosZSW1 OR W#16#01;
       ELSE
         #swEPosZSW1 := #swEPosZSW1 AND W#16#FFFE;
       END_IF;

       // EPOS-Wort-1 Bit 01 --> 1 = Active traversing block bit 1
       //IF #sxRecvBuf.sxEPosZSW1.ActTrvBit1 THEN
       IF #sxRecvBuf.EPosZSW1.%X1 THEN
         #swEPosZSW1 := #swEPosZSW1 OR W#16#02;
       ELSE
         #swEPosZSW1 := #swEPosZSW1 AND W#16#FFFD;
       END_IF;

       // EPOS-Wort-1 Bit 02 --> 1 = Active traversing block bit 2
       //IF #sxRecvBuf.sxEPosZSW1.ActTrvBit2 THEN
       IF #sxRecvBuf.EPosZSW1.%X2 THEN
         #swEPosZSW1 := #swEPosZSW1 OR W#16#04;
       ELSE
         #swEPosZSW1 := #swEPosZSW1 AND W#16#FFFB;
       END_IF;

       // EPOS-Wort-1 Bit 03 --> 1 = Active traversing block bit 3
       //IF #sxRecvBuf.sxEPosZSW1.ActTrvBit3 THEN
       IF #sxRecvBuf.EPosZSW1.%X3 THEN
         #swEPosZSW1 := #swEPosZSW1 OR W#16#08;
       ELSE
         #swEPosZSW1 := #swEPosZSW1 AND W#16#FFF7;
       END_IF;

       // EPOS-Wort-1 Bit 04 --> 1 = Active traversing block bit 4 
       //IF #sxRecvBuf.sxEPosZSW1.ActTrvBit4 THEN
       IF #sxRecvBuf.EPosZSW1.%X4 THEN
         #swEPosZSW1 := #swEPosZSW1 OR W#16#10;
       ELSE
         #swEPosZSW1 := #swEPosZSW1 AND W#16#FFEF;
       END_IF;

       // EPOS-Wort-1 Bit 05 --> 1 = Active traversing block bit 5
       //IF #sxRecvBuf.sxEPosZSW1.ActTrvBit5 THEN
       IF #sxRecvBuf.EPosZSW1.%X5 THEN
         #swEPosZSW1 := #swEPosZSW1 OR W#16#20;
       ELSE
         #swEPosZSW1 := #swEPosZSW1 AND W#16#FFDF;
       END_IF;

       // EPOS-Wort-1 Bit 08 --> 1 = STOP cam minus active
       //IF #sxRecvBuf.sxEPosZSW1.StpCamMinAct THEN
       IF #sxRecvBuf.EPosZSW1.%X8 THEN
         #swEPosZSW1 := #swEPosZSW1 OR W#16#100;
       ELSE
         #swEPosZSW1 := #swEPosZSW1 AND W#16#FEFF;
       END_IF;

       // EPOS-Wort-1 Bit 09 --> 1 = STOP cam plus active
       //IF #sxRecvBuf.sxEPosZSW1.StpCamPlsAct THEN
       IF #sxRecvBuf.EPosZSW1.%X9 THEN
         #swEPosZSW1 := #swEPosZSW1 OR W#16#200;
       ELSE
         #swEPosZSW1 := #swEPosZSW1 AND W#16#FDFF;
       END_IF;

       // EPOS-Wort-1 Bit 10 --> 1 = Jogging active
       //IF #sxRecvBuf.sxEPosZSW1.JogAct THEN
       IF #sxRecvBuf.EPosZSW1.%X10 THEN
         #swEPosZSW1 := #swEPosZSW1 OR W#16#400;
       ELSE
         #swEPosZSW1 := #swEPosZSW1 AND W#16#FBFF;
       END_IF;

       // EPOS-Wort-1 Bit 11 --> 1 = Reference point approach active
       //IF #sxRecvBuf.sxEPosZSW1.RefAct THEN
       IF #sxRecvBuf.EPosZSW1.%X11 THEN
         #swEPosZSW1 := #swEPosZSW1 OR W#16#800;
       ELSE
         #swEPosZSW1 := #swEPosZSW1 AND W#16#F7FF;
       END_IF;

       // Anstossen des fliegenden Referenzieren prüfen, wenn die Rückmeldung fehlt dann wiederholen
       //IF NOT #sxRecvBuf.sxEPosZSW1.FlyRefAct AND #sbRefTyp AND #sxSendBuf.sxSTW1.RefStart THEN
       IF NOT #sxRecvBuf.EPosZSW1.%X12 AND #sbRefTyp AND #sxSendBuf.STW1.%X11 THEN

         // Wiederholung anstossen 
         IF #siRefActRetry < #siRetryMax THEN
           #siRefActRetry := #siRefActRetry + 1;

           // Referenzieren starten wieder wegnehmen
           //#sxSendBuf.sxSTW1.RefStart := False;
           #sxSendBuf.STW1.%X11 := False;
         ELSE

           // Fehlermeldung
           #swStatus := 16#8403;
           #Error := True;
         END_IF;
       ELSE

         // Fehler wieder zurücknehmen, wenn er mal ausgelöst wurde
         IF #swStatus = 16#8403 THEN
           #swStatus := 16#7002;
           #Error := False;
         END_IF;
         // Zähler zurücksetzen bei Rückmeldung fliegendes Referenzieren jetzt aktiviert oder bei Abwahl der Funktion
         IF (#sxRecvBuf.EPosZSW1.%X12 AND #sbRefTyp AND #sxSendBuf.STW1.%X11) OR NOT #FlyRef THEN
           #siRefActRetry := 0;
         END_IF;
       END_IF;

       // EPOS-Wort-1 Bit 12 --> 1 = Flying referencing active
       //IF #sxRecvBuf.sxEPosZSW1.FlyRefAct THEN
       IF #sxRecvBuf.EPosZSW1.%X12 THEN
         #swEPosZSW1 := #swEPosZSW1 OR W#16#1000;
       ELSE
         #swEPosZSW1 := #swEPosZSW1 AND W#16#EFFF;
       END_IF;

       // EPOS-Wort-1 Bit 13 --> 1 = Traversing block active
       //IF #sxRecvBuf.sxEPosZSW1.TrvBlAct THEN
       IF #sxRecvBuf.EPosZSW1.%X13 THEN
         #swEPosZSW1 := #swEPosZSW1 OR W#16#2000;
       ELSE
         #swEPosZSW1 := #swEPosZSW1 AND W#16#DFFF;
       END_IF;

       // EPOS-Wort-1 Bit 14 --> 1 = MDI setup active
       //IF #sxRecvBuf.sxEPosZSW1.MdiStupAct THEN
       IF #sxRecvBuf.EPosZSW1.%X14 THEN
         #swEPosZSW1 := #swEPosZSW1 OR W#16#4000;
       ELSE
         #swEPosZSW1 := #swEPosZSW1 AND W#16#BFFF;
       END_IF;

       // EPOS-Wort-1 Bit 15 --> 1 = MDI positing active
       //IF #sxRecvBuf.sxEPosZSW1.MdiPosAct THEN
       IF #sxRecvBuf.EPosZSW1.%X15 THEN
         #swEPosZSW1 := #swEPosZSW1 OR W#16#8000;
       ELSE
         #swEPosZSW1 := #swEPosZSW1 AND W#16#7FFF;
       END_IF;

       // EPOS_ZSW2 
       // EPOS-Wort-2 Bit 00 --> 1 = Tracking mode active
       //IF #sxRecvBuf.sxEPosZSW2.TrkModeAct THEN
       IF #sxRecvBuf.EPosZSW2.%X0 THEN
         #swEPosZSW2 := #swEPosZSW2 OR W#16#01;
       ELSE
         #swEPosZSW2 := #swEPosZSW2 AND W#16#FFFE;
       END_IF;

       // EPOS-Wort-2 Bit 01 --> 1 = Velocity limit active
       //IF #sxRecvBuf.sxEPosZSW2.VeloLimAct THEN
       IF #sxRecvBuf.EPosZSW2.%X1 THEN
         #swEPosZSW2 := #swEPosZSW2 OR W#16#02;
       ELSE
         #swEPosZSW2 := #swEPosZSW2 AND W#16#FFFD;
       END_IF;

       // EPOS-Wort-2 Bit 02 --> 1 = Setpoint static
       //IF #sxRecvBuf.sxEPosZSW2.SetPStat THEN
       IF #sxRecvBuf.EPosZSW2.%X2 THEN
         #swEPosZSW2 := #swEPosZSW2 OR W#16#04;
       ELSE
         #swEPosZSW2 := #swEPosZSW2 AND W#16#FFFB;
       END_IF;

       // EPOS-Wort-2 Bit 03 --> 1 = Printmark outside outer window
       //IF #sxRecvBuf.sxEPosZSW2.PrnMrkOut THEN
       IF #sxRecvBuf.EPosZSW2.%X3 THEN
         #swEPosZSW2 := #swEPosZSW2 OR W#16#08;
       ELSE
         #swEPosZSW2 := #swEPosZSW2 AND W#16#FFF7;
       END_IF;

       // EPOS-Wort-2 Bit 04 --> 1 = Axis forwards
       //IF #sxRecvBuf.sxEPosZSW2.FWD THEN
       IF #sxRecvBuf.EPosZSW2.%X4 THEN
         #swEPosZSW2 := #swEPosZSW2 OR W#16#10;
       ELSE
         #swEPosZSW2 := #swEPosZSW2 AND W#16#FFEF;
       END_IF;

       // EPOS-Wort-2 Bit 05 --> 1 = Axis backwards
       //IF #sxRecvBuf.sxEPosZSW2.BWD THEN
       IF #sxRecvBuf.EPosZSW2.%X5 THEN
         #swEPosZSW2 := #swEPosZSW2 OR W#16#20;
       ELSE
         #swEPosZSW2 := #swEPosZSW2 AND W#16#FFDF;
       END_IF;

       // EPOS-Wort-2 Bit 06 --> 1 = Software limit switch minus active
       //IF #sxRecvBuf.sxEPosZSW2.SftSwMinAct THEN
       IF #sxRecvBuf.EPosZSW2.%X6 THEN
         #swEPosZSW2 := #swEPosZSW2 OR W#16#40;
       ELSE
         #swEPosZSW2 := #swEPosZSW2 AND W#16#FFBF;
       END_IF;

       // EPOS-Wort-2 Bit 07 --> 1 = Software limit switch plus active
       //IF #sxRecvBuf.sxEPosZSW2.SftSwPlsAct THEN
       IF #sxRecvBuf.EPosZSW2.%X7 THEN
         #swEPosZSW2 := #swEPosZSW2 OR W#16#80;
       ELSE
         #swEPosZSW2 := #swEPosZSW2 AND W#16#FF7F;
       END_IF;

       // EPOS-Wort-2 Bit 08 --> 1 = Position actual value <= cam position 1
       //IF #sxRecvBuf.sxEPosZSW2.PosSmCam1 THEN
       IF #sxRecvBuf.EPosZSW2.%X8 THEN
         #swEPosZSW2 := #swEPosZSW2 OR W#16#100;
       ELSE
         #swEPosZSW2 := #swEPosZSW2 AND W#16#FEFF;
       END_IF;

       // EPOS-Wort-2 Bit 09 --> 1 = Position actual value <= cam position 2
       //IF #sxRecvBuf.sxEPosZSW2.PosSmCam2 THEN
       IF #sxRecvBuf.EPosZSW2.%X9 THEN
         #swEPosZSW2 := #swEPosZSW2 OR W#16#200;
       ELSE
         #swEPosZSW2 := #swEPosZSW2 AND W#16#FDFF;
       END_IF;

       // EPOS-Wort-2 Bit 10 --> 1 = Direct output 1 via traversing block
       //IF #sxRecvBuf.sxEPosZSW2.TrvOut1 THEN
       IF #sxRecvBuf.EPosZSW2.%X10 THEN
         #swEPosZSW2 := #swEPosZSW2 OR W#16#400;
       ELSE
         #swEPosZSW2 := #swEPosZSW2 AND W#16#FBFF;
       END_IF;

       // EPOS-Wort-2 Bit 11 --> 1 = Direct output 2 via traversing block
       //IF #sxRecvBuf.sxEPosZSW2.TrvOut2 THEN
       IF #sxRecvBuf.EPosZSW2.%X11 THEN
         #swEPosZSW2 := #swEPosZSW2 OR W#16#800;
       ELSE
         #swEPosZSW2 := #swEPosZSW2 AND W#16#F7FF;
       END_IF;

       // EPOS-Wort-2 Bit 12 --> 1 = Fixed STOP reached
       //IF #sxRecvBuf.sxEPosZSW2.FxStpRd THEN
       IF #sxRecvBuf.EPosZSW2.%X12 THEN
         #swEPosZSW2 := #swEPosZSW2 OR W#16#1000;
       ELSE
         #swEPosZSW2 := #swEPosZSW2 AND W#16#EFFF;
       END_IF;

       // EPOS-Wort-2 Bit 13 --> 1 = Fixed STOP clamping torque reached
       //IF #sxRecvBuf.sxEPosZSW2.FxStpTrRd THEN
       IF #sxRecvBuf.EPosZSW2.%X13 THEN
         #swEPosZSW2 := #swEPosZSW2 OR W#16#2000;
       ELSE
         #swEPosZSW2 := #swEPosZSW2 AND W#16#DFFF;
       END_IF;

       // EPOS-Wort-2 Bit 14 --> 1 = Traversing fixed STOP active
       //IF #sxRecvBuf.sxEPosZSW2.TrvFxStpAct THEN
       IF #sxRecvBuf.EPosZSW2.%X14 THEN
         #swEPosZSW2 := #swEPosZSW2 OR W#16#4000;
       ELSE
         #swEPosZSW2 := #swEPosZSW2 AND W#16#BFFF;
       END_IF;

       // EPOS-Wort-2 Bit 15 --> 1 = Traversing command active
       //IF #sxRecvBuf.sxEPosZSW2.CmdAct THEN
       IF #sxRecvBuf.EPosZSW2.%X15 THEN
         #swEPosZSW2 := #swEPosZSW2 OR W#16#8000;
       ELSE
         #swEPosZSW2 := #swEPosZSW2 AND W#16#7FFF;
       END_IF;

       #sbReady := #sxRecvBuf.ZSW1.%X1;

       #AxisEnabled := #sxRecvBuf.ZSW1.%X2;
       #sbIOp := #sxRecvBuf.ZSW1.%X2;

       #AxisError := #sxRecvBuf.ZSW1.%X3;
       #sbFault := #sxRecvBuf.ZSW1.%X3;

       #AxisWarn := #sxRecvBuf.ZSW1.%X7;
       #sbAlarm := #sxRecvBuf.ZSW1.%X7;

       #AxisPosOk := #sxRecvBuf.ZSW1.%X10;
       #AxisRef := #sxRecvBuf.ZSW1.%X11;
       #AxisSpFixed := #sxRecvBuf.ZSW1.%X13;

       #sbAccel := #sxRecvBuf.ZSW1.%X14;
       #sbDecel := #sxRecvBuf.ZSW1.%X15;

       #ActVelocity := DWORD_TO_DINT(#sxRecvBuf.Velocity);
       #ActPosition := DWORD_TO_DINT(#sxRecvBuf.Position);
       #ActMode := #ModePos;
       #ActWarn := #sxRecvBuf.WarnNr;
       #ActFault := #sxRecvBuf.ErrNr;

       #Lockout := #sxRecvBuf.ZSW1.%X6;
     END_IF;
   ELSE

     // Fehler
     #Error := TRUE;
     #swStatus := 16#8601;

   END_IF;

   // Initialisierung von Ausg㭧en
   #Status := #swStatus;
   #EPosZSW1 := #swEPosZSW1;
   #EPosZSW2 := #swEPosZSW2;
END_FUNCTION_BLOCK

ORGANIZATION_BLOCK "Main"   // OB1, LAD, ProgramCycle
TITLE = "Main Program Sweep (Cycle)"
{ S7_Optimized_Access := 'TRUE' }
VERSION : 0.1
   VAR_INPUT
      Initial_Call : Bool;   // Initial call of this OB
      Remanence : Bool;   // =True, if remanent data are available
   END_VAR
BEGIN

REGION Network 1
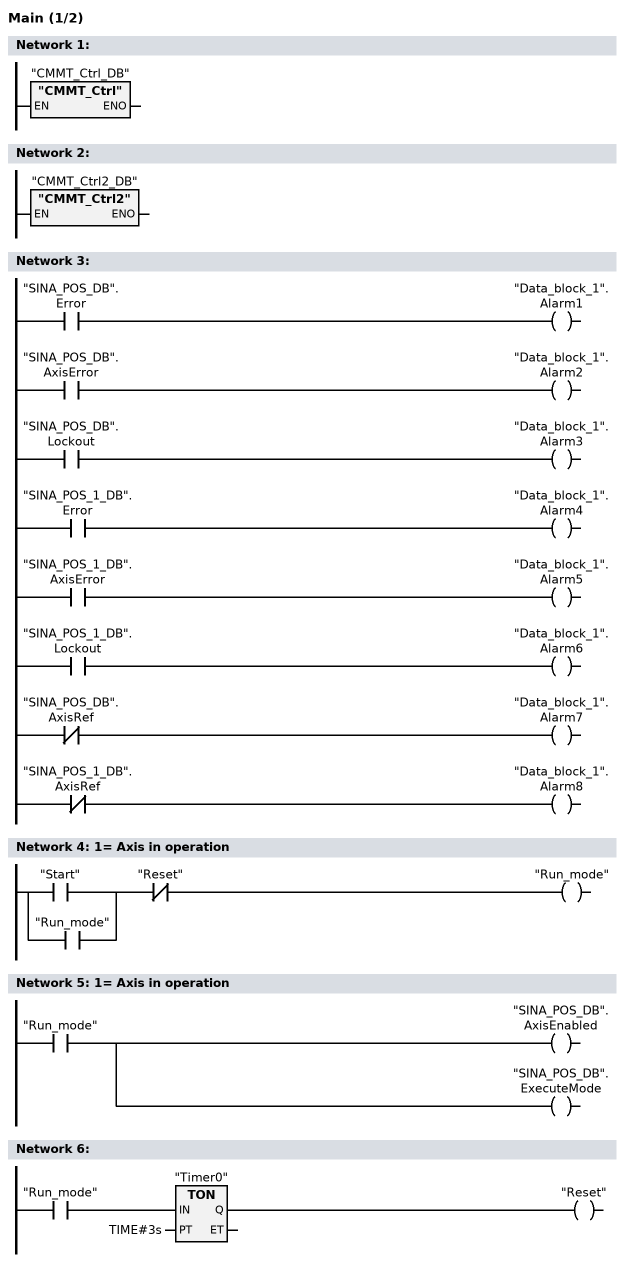
   RUNG wire#powerrail
      "CMMT_Ctrl_DB"()
   END_RUNG
   // the same network as SCL:
   "CMMT_Ctrl_DB"();   // "CMMT_Ctrl"
END_REGION

REGION Network 2
   RUNG wire#powerrail
      "CMMT_Ctrl2_DB"()
   END_RUNG
   // the same network as SCL:
   "CMMT_Ctrl2_DB"();   // "CMMT_Ctrl2"
END_REGION

REGION Network 3
   RUNG wire#powerrail
      Contact( "SINA_POS_DB".Error )
      Coil( "Data_block_1".Alarm1 )
   END_RUNG
   RUNG wire#powerrail
      Contact( "SINA_POS_DB".AxisError )
      Coil( "Data_block_1".Alarm2 )
   END_RUNG
   RUNG wire#powerrail
      Contact( "SINA_POS_DB".Lockout )
      Coil( "Data_block_1".Alarm3 )
   END_RUNG
   RUNG wire#powerrail
      Contact( "SINA_POS_1_DB".Error )
      Coil( "Data_block_1".Alarm4 )
   END_RUNG
   RUNG wire#powerrail
      Contact( "SINA_POS_1_DB".AxisError )
      Coil( "Data_block_1".Alarm5 )
   END_RUNG
   RUNG wire#powerrail
      Contact( "SINA_POS_1_DB".Lockout )
      Coil( "Data_block_1".Alarm6 )
   END_RUNG
   RUNG wire#powerrail
      I_Contact( "SINA_POS_DB".AxisRef )
      Coil( "Data_block_1".Alarm7 )
   END_RUNG
   RUNG wire#powerrail
      I_Contact( "SINA_POS_1_DB".AxisRef )
      Coil( "Data_block_1".Alarm8 )
   END_RUNG
   // the same network as SCL:
   "Data_block_1".Alarm1 := "SINA_POS_DB".Error;
   "Data_block_1".Alarm2 := "SINA_POS_DB".AxisError;
   "Data_block_1".Alarm3 := "SINA_POS_DB".Lockout;
   "Data_block_1".Alarm4 := "SINA_POS_1_DB".Error;
   "Data_block_1".Alarm5 := "SINA_POS_1_DB".AxisError;
   "Data_block_1".Alarm6 := "SINA_POS_1_DB".Lockout;
   "Data_block_1".Alarm7 := NOT "SINA_POS_DB".AxisRef;
   "Data_block_1".Alarm8 := NOT "SINA_POS_1_DB".AxisRef;
END_REGION

REGION Network 4: 1= Axis in operation
   RUNG wire#powerrail
      Contact( "Start" )
      wire#w1
      I_Contact( "Reset" )
      Coil( "Run_mode" )
   END_RUNG
   RUNG wire#powerrail
      Contact( "Run_mode" )
   END_RUNG wire#w1
   // the same network as SCL:
   "Run_mode" := ("Start" OR "Run_mode") AND NOT "Reset";
END_REGION

REGION Network 5: 1= Axis in operation
   RUNG wire#powerrail
      Contact( "Run_mode" )
      wire#w1
      Coil( "SINA_POS_DB".AxisEnabled )
   END_RUNG
   RUNG wire#w1
      Coil( "SINA_POS_DB".ExecuteMode )
   END_RUNG
   // the same network as SCL:
   "SINA_POS_DB".AxisEnabled := "Run_mode";
   "SINA_POS_DB".ExecuteMode := "Run_mode";
END_REGION

REGION Network 6
   "Timer0".TON(IN := "Run_mode", PT := TIME#3s);
   "Reset" := "Timer0".Q;
END_REGION

REGION Network 7: 1 = Acknowledge of errors
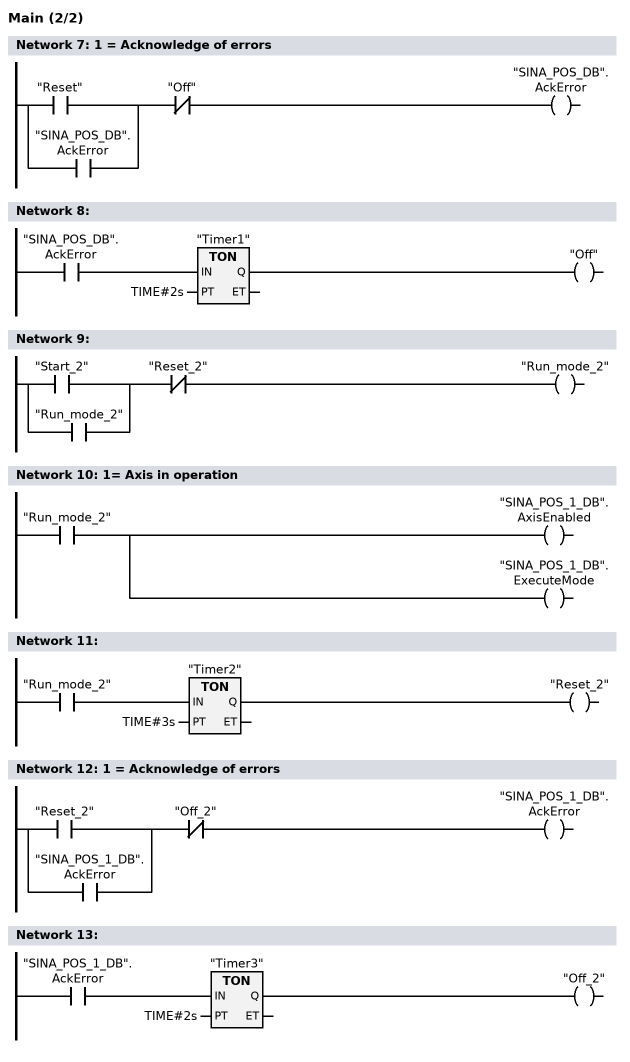
   RUNG wire#powerrail
      Contact( "Reset" )
      wire#w1
      I_Contact( "Off" )
      Coil( "SINA_POS_DB".AckError )
   END_RUNG
   RUNG wire#powerrail
      Contact( "SINA_POS_DB".AckError )
   END_RUNG wire#w1
   // the same network as SCL:
   "SINA_POS_DB".AckError := ("Reset" OR "SINA_POS_DB".AckError) AND NOT "Off";
END_REGION

REGION Network 8
   "Timer1".TON(IN := "SINA_POS_DB".AckError, PT := TIME#2s);
   "Off" := "Timer1".Q;
END_REGION

REGION Network 9
   RUNG wire#powerrail
      Contact( "Start_2" )
      wire#w1
      I_Contact( "Reset_2" )
      Coil( "Run_mode_2" )
   END_RUNG
   RUNG wire#powerrail
      Contact( "Run_mode_2" )
   END_RUNG wire#w1
   // the same network as SCL:
   "Run_mode_2" := ("Start_2" OR "Run_mode_2") AND NOT "Reset_2";
END_REGION

REGION Network 10: 1= Axis in operation
   RUNG wire#powerrail
      Contact( "Run_mode_2" )
      wire#w1
      Coil( "SINA_POS_1_DB".AxisEnabled )
   END_RUNG
   RUNG wire#w1
      Coil( "SINA_POS_1_DB".ExecuteMode )
   END_RUNG
   // the same network as SCL:
   "SINA_POS_1_DB".AxisEnabled := "Run_mode_2";
   "SINA_POS_1_DB".ExecuteMode := "Run_mode_2";
END_REGION

REGION Network 11
   "Timer2".TON(IN := "Run_mode_2", PT := TIME#3s);
   "Reset_2" := "Timer2".Q;
END_REGION

REGION Network 12: 1 = Acknowledge of errors
   RUNG wire#powerrail
      Contact( "Reset_2" )
      wire#w1
      I_Contact( "Off_2" )
      Coil( "SINA_POS_1_DB".AckError )
   END_RUNG
   RUNG wire#powerrail
      Contact( "SINA_POS_1_DB".AckError )
   END_RUNG wire#w1
   // the same network as SCL:
   "SINA_POS_1_DB".AckError := ("Reset_2" OR "SINA_POS_1_DB".AckError) AND NOT "Off_2";
END_REGION

REGION Network 13
   "Timer3".TON(IN := "SINA_POS_1_DB".AckError, PT := TIME#2s);
   "Off_2" := "Timer3".Q;
END_REGION
END_ORGANIZATION_BLOCK

(* ===== HMI "HMI_RT_1" =====
system functions are stored by id; their names below are inferred from use
connection "HMI_Connection_1": ETHERNET, SMART_S7_1200_OMS

HMI tags "Default tag table"
   "Tag_ScreenNumber" : UInt, internal
   "HMI_Tag_1" : Int, internal
   "SINA_POS_DB_ModePos" : Int = PLC SINA_POS_DB.ModePos, 1 s
   "SINA_POS_DB_EnableAxis" : Bool = PLC SINA_POS_DB.EnableAxis, 1 s
   "SINA_POS_DB_ExecuteMode" : Bool = PLC SINA_POS_DB.ExecuteMode, 1 s
   "SINA_POS_DB_Velocity" : DInt = PLC SINA_POS_DB.Velocity, 1 s
   "SINA_POS_DB_Position" : DInt = PLC SINA_POS_DB.Position, 1 s
   "SINA_POS_DB_AckError" : Bool = PLC SINA_POS_DB.AckError, 1 s
   "SINA_POS_DB_1_Velocity" : DInt = PLC SINA_POS_1_DB.Velocity, 1 s
   "SINA_POS_DB_1_Position" : DInt = PLC SINA_POS_1_DB.Position, 1 s
   "SINA_POS_DB_1_ModePoss" : Int = PLC SINA_POS_1_DB.ModePos, 1 s
   "SINA_POS_DB_1_ExecuteMode" : Bool = PLC SINA_POS_1_DB.ExecuteMode, 1 s
   "SINA_POS_DB_1_EnableAxis" : Bool = PLC SINA_POS_1_DB.EnableAxis, 1 s
   "SINA_POS_DB_1_AckError" : Bool = PLC SINA_POS_1_DB.AckError, 1 s
   "SINA_POS_DB_ERROR" : Int AT %DB5.DBW0, 1 s
   "SINA_POS_DB_ERROR(1)" : Bool = PLC SINA_POS_DB.Error, 1 s
   "Set reff" : Bool = PLC Start AT %I0.1, 1 s
   "Set reff_2" : Bool = PLC Start_2 AT %M0.5, 1 s

discrete alarms
   1: 'Error Axis', class Errors, trigger "SINA_POS_DB_ERROR" bit 9
   2: 'Error', class Errors, trigger "SINA_POS_DB_ERROR" bit 8
   3: 'Locked', class Errors, trigger "SINA_POS_DB_ERROR" bit 10
   4: 'Error Axis Motor 2', class Errors, trigger "SINA_POS_DB_ERROR" bit 12
   5: 'Error Motor 2', class Errors, trigger "SINA_POS_DB_ERROR" bit 11
   6: 'Locked Motor 2', class Errors, trigger "SINA_POS_DB_ERROR" bit 13
   7: 'Axis Reff off', class Errors, trigger "SINA_POS_DB_ERROR" bit 14
   8: 'Axis Reff off Motor 2', class Errors, trigger "SINA_POS_DB_ERROR" bit 15

analog alarms
   1: '', class Errors

text list "Mode pos": 1 '1'; 2 '2'; 7 '7'; 4 '4'; 5 '5'

Template "Template_1" 800x480
   Button "Exit" at 714,429 size 71x50; TextOff 'Exit'; PictureOff "ExitRuntime_KTP700_Basic_PN_TR"; PictureOn "ExitRuntime_KTP700_Basic_PN_TR"
      on Release: StopRuntime(0)
   Button "Template_Button" at 614,429 size 71x50; TextOff 'Text'
   Button "Template_Button_1" at 514,429 size 71x50; TextOff 'Text'
   Button "Template_Button_2" at 414,429 size 71x50; TextOff 'Text'
   Button "Template_Button_3" at 314,429 size 71x50; TextOff 'Text'
   Button "Template_Button_4" at 214,429 size 71x50; TextOff 'Text'
   Button "Alarms" at 114,429 size 71x50; TextOff 'Alarms'; PictureOff "AlarmDisplay_KTP700_Basic_PN_TR"; PictureOn "AlarmDisplay_KTP700_Basic_PN_TR"
      on Release: function_ef3f5d25("Alarm window_Pending", -1)
   Button "Start screen" at 14,429 size 71x50; TextOff 'Start screen'; PictureOff "NavigateHome_KTP700_Basic_PN_TR"; PictureOn "NavigateHome_KTP700_Basic_PN_TR"
      on Release: ActivateScreen("Root screen", 0)
   Button "Template_Button_5" at 727,52 size 71x50; TextOff 'Text'
   Button "Template_Button_6" at 727,106 size 71x50; TextOff 'Text'
   Button "Template_Button_7" at 727,159 size 71x50; TextOff 'Text'
   Button "Template_Button_8" at 727,213 size 71x50; TextOff 'Text'
   Button "Template_Button_9" at 727,267 size 71x50; TextOff 'Text'
   Button "Template_Button_10" at 727,321 size 71x50; TextOff 'Text'
   Button "Template_Button_11" at 727,374 size 71x50; TextOff 'Text'
   SymbolicIOField "Symbolic_IO_Field_Screen" at 93,9 size 600x33; TextOff '0'; TextOn '1'; TextList "TextList_ScreenNames"
      ProcessValue <- "Tag_ScreenNumber"
      on Change: ActivateScreenByNumber("Tag_ScreenNumber", 0)
   DateTimeField "HmiScreenItemData" at 695,25 size 105x25
   DateTimeField "HmiScreenItemData_1" at 695,0 size 105x25
   GraphicView "Logo" at 0,0 size 91x51; Picture "Logo of HMI_1"

screen "Root screen" 800x480, template "Template_1"
   on GenerateScreen: SetTag("Tag_ScreenNumber", 1)
   Button "HmiScreenItemData_2" at 26,117 size 159x47; TextOff 'System screens'; PictureOff "Navigates to System screens for KTP700 Basic+ PN 15.1.0.0"; PictureOn "Navigates to System screens for KTP700 Basic+ PN 15.1.0.0"
      on Release: ActivateScreen("System screens", 0)
   Switch "Template_Switch_2" at 370,300 size 64x32; TextOn 'ON'; CaptionText 'Switch'; TextOff 'OFF'
      ProcessValue <- "SINA_POS_DB_EnableAxis"
   SymbolicIOField "Template_Symbolic I/O field_1" at 608,300 size 96x32; TextOn '1'; TextOff '0'; TextList "Mode pos"
      ProcessValue <- "SINA_POS_DB_ModePos"
   TextField "Template_Text field_1" at 628,257 size 49x23; Text 'Mode'
   TextField "Template_Text field_2" at 343,257 size 98x23; Text 'Enable axis'
   IOField "Template_I/O field_1" at 221,301 size 96x35; FormatPattern 99999
      ProcessValue <- "SINA_POS_DB_Velocity"
   IOField "Template_I/O field_2" at 88,301 size 96x32; FormatPattern 99999
      ProcessValue <- "SINA_POS_DB_Position"
   TextField "Template_Text field_4" at 235,262 size 63x23; Text 'Velociy'
   TextField "Template_Text field_5" at 98,264 size 71x23; Text 'Position'
   Button "HmiScreenItemData_5" at 26,177 size 159x47; TextOn 'Motor 2'; TextOff 'Motor 2'; PictureOn "Navigates to Project information for KTP700 Basic+ PN 15.1.0.0"; PictureOff "Navigates to Project information for KTP700 Basic+ PN 15.1.0.0"
      on Release: ActivateScreen("Root screen_1", 0)
   Button "Button_1" at 524,199 size 177x32; TextOff 'Aknowladge Error'
      on Press: function_b14e0dd5("SINA_POS_DB_AckError", 0); function_b14e0dd5("SINA_POS_DB_ExecuteMode", 0); function_b14e0dd5("SINA_POS_DB_EnableAxis", 0)
   Button "Button_2" at 462,300 size 126x32; TextOff 'Execute Mode'
      on Press: function_b14e0dd5("SINA_POS_DB_ExecuteMode", 0)
   Button "Button_3" at 350,199 size 126x32; TextOff 'Set Axis'
      on Press: function_b14e0dd5("Set reff", 0)

screen "System screens" 800x480, template "Template_1"
   on GenerateScreen: SetTag("Tag_ScreenNumber", 4)
   Button "Back" at 1,52 size 159x47; TextOff 'Back'
      on Release: ActivateScreen("Root screen", 0)
   Button "HmiScreenItemData" at 36,146 size 159x47; TextOff 'SIMATIC PLC system diagnos...'; PictureOff "Navigates to SIMATIC PLC system diagnostics for KTP700 Basic+ PN 15.1.0.0"; PictureOn "Navigates to SIMATIC PLC system diagnostics for KTP700 Basic+ PN 15.1.0.0"
      on Release: ActivateScreen("SIMATIC PLC system diagnostics", 0)
   Button "HmiScreenItemData_1" at 36,205 size 159x47; TextOff 'Project information'; PictureOff "Navigates to Project information for KTP700 Basic+ PN 15.1.0.0"; PictureOn "Navigates to Project information for KTP700 Basic+ PN 15.1.0.0"
      on Release: ActivateScreen("Project information", 0)
   Button "HmiScreenItemData_2" at 36,264 size 159x47; TextOff 'User administration'; PictureOff "Navigates to User administration for KTP700 Basic+ PN 15.1.0.0"; PictureOn "Navigates to User administration for KTP700 Basic+ PN 15.1.0.0"
      on Release: ActivateScreen("User administration", 0)
   Button "HmiScreenItemData_3" at 36,323 size 159x47; TextOff 'System information'; PictureOff "Navigates to System information for KTP700 Basic+ PN 15.1.0.0"; PictureOn "Navigates to System information for KTP700 Basic+ PN 15.1.0.0"
      on Release: ActivateScreen("System information", 0)
   Button "HmiScreenItemData_4" at 207,146 size 159x47; TextOff 'Different jobs'; PictureOff "Navigates to Different jobs for KTP700 Basic+ PN 15.1.0.0"; PictureOn "Navigates to Different jobs for KTP700 Basic+ PN 15.1.0.0"
      on Release: ActivateScreen("Different jobs", 0)

screen "SIMATIC PLC system diagnostics" 800x480, template "Template_1"
   on GenerateScreen: SetTag("Tag_ScreenNumber", 5)
   SysDiagControl "HmiScreenItemData" at 1,100 size 724x321
   Button "Back" at 1,52 size 159x47; TextOff 'Back'
      on Release: ActivateScreen("System screens", 0)

screen "Project information" 800x480, template "Template_1"
   on GenerateScreen: SetTag("Tag_ScreenNumber", 6)
   TextField "HmiScreenItemData" at 35,102 size 171x28; Text 'Project name:'
   TextField "HmiScreenItemData_1" at 241,102 size 452x28; Text 'Project1'
   TextField "HmiScreenItemData_2" at 35,132 size 171x28; Text 'Created on:'
   TextField "HmiScreenItemData_3" at 241,132 size 452x28; Text '8/20/2021 5:52:06 PM'
   TextField "HmiScreenItemData_4" at 35,162 size 171x28; Text 'Author:'
   TextField "HmiScreenItemData_5" at 241,162 size 452x28; Text 'diego'
   TextField "HmiScreenItemData_6" at 35,192 size 171x28; Text 'Description:'
   TextField "HmiScreenItemData_7" at 241,192 size 452x28; Text '(not configured)'
   Button "Back" at 1,52 size 159x47; TextOff 'Back'
      on Release: ActivateScreen("System screens", 0)

screen "User administration" 800x480, template "Template_1"
   on GenerateScreen: SetTag("Tag_ScreenNumber", 7)
   UserView "HmiScreenItemData" at 1,100 size 724x321
   Button "Back" at 1,52 size 159x47; TextOff 'Back'
      on Release: ActivateScreen("System screens", 0)

screen "System information" 800x480, template "Template_1"
   on GenerateScreen: SetTag("Tag_ScreenNumber", 8)
   TextField "HmiScreenItemData" at 35,102 size 171x28; Text 'HMI device type:'
   TextField "HmiScreenItemData_1" at 241,102 size 452x28; Text 'KTP700 Basic+ PN 15.1.0.0'
   TextField "HmiScreenItemData_2" at 35,132 size 171x28; Text 'Connection:'
   TextField "HmiScreenItemData_3" at 241,132 size 452x28; Text 'PROFINET (X1)'
   TextField "HmiScreenItemData_4" at 35,162 size 171x28; Text 'PLC:'
   TextField "HmiScreenItemData_5" at 241,162 size 452x28; Text 'SIMATIC S7 1200'
   Button "Back" at 1,52 size 159x47; TextOff 'Back'
      on Release: ActivateScreen("System screens", 0)

screen "Different jobs" 800x480, template "Template_1"
   on GenerateScreen: SetTag("Tag_ScreenNumber", 9)
   Button "Online" at 36,146 size 159x47; TextOff 'Online'
      on Release: function_bb44b551(0)
   Button "Offline" at 36,205 size 159x47; TextOff 'Offline'
      on Release: function_bb44b551(1)
   Button "Transfer" at 36,264 size 159x47; TextOff 'Transfer'
      on Release: function_bb44b551(2)
   Button "Toggle language" at 36,323 size 159x47; TextOff 'Toggle language'
      on Release: function_fb9197e8(-1)
   Button "Stop Runtime" at 207,146 size 159x47; TextOff 'Stop Runtime'
      on Release: StopRuntime(0)
   Button "Back" at 1,52 size 159x47; TextOff 'Back'
      on Release: ActivateScreen("System screens", 0)

screen "Root screen_1" 800x480, template "Template_1"
   on GenerateScreen: SetTag("Tag_ScreenNumber", 2)
   Switch "Template_Switch_2" at 370,300 size 64x32; TextOn 'ON'; CaptionText 'Switch'; TextOff 'OFF'
      ProcessValue <- "SINA_POS_DB_1_EnableAxis"
   SymbolicIOField "Template_Symbolic I/O field_1" at 624,300 size 96x32; TextOn '1'; TextOff '0'; TextList "Mode pos"
      ProcessValue <- "SINA_POS_DB_1_ModePoss"
   TextField "Template_Text field_1" at 638,262 size 49x23; Text 'Mode'
   TextField "Template_Text field_2" at 343,257 size 98x23; Text 'Enable axis'
   IOField "Template_I/O field_1" at 221,301 size 96x35; FormatPattern 99999
      ProcessValue <- "SINA_POS_DB_1_Velocity"
   IOField "Template_I/O field_2" at 88,301 size 96x32; FormatPattern 99999
      ProcessValue <- "SINA_POS_DB_1_Position"
   TextField "Template_Text field_4" at 238,258 size 63x23; Text 'Velociy'
   TextField "Template_Text field_5" at 101,252 size 71x23; Text 'Position'
   Button "Back" at 1,52 size 159x47; TextOn 'Back'; TextOff 'Back'
      on Release: ActivateScreen("Root screen", 0)
   Button "Button_1" at 524,199 size 177x32; TextOff 'Aknowladge Error'
      on Press: function_b14e0dd5("SINA_POS_DB_AckError", 0); function_b14e0dd5("SINA_POS_DB_1_ExecuteMode", 0); function_b14e0dd5("SINA_POS_DB_1_EnableAxis", 0)
   Button "Button_2" at 462,300 size 126x32; TextOff 'Execute Mode'
      on Press: function_b14e0dd5("SINA_POS_DB_1_ExecuteMode", 0)
   Button "Button_3" at 350,199 size 126x32; TextOff 'Set Axis'
      on Press: function_b14e0dd5("Set reff_2", 0)
*)